FUNCTION F_CAMERA_Evaluation : BOOL
VAR_INPUT
	nExpectedResp		: INT;
	nCodesRead			: INT;
	bResetEval		  	: BOOL;
END_VAR
VAR_IN_OUT
	aCodeData			: ARRAY[1..cMAX_CAMERA_PROG_NUMBER] OF ST_CAMERA_CodeData;
	stCameraEvaluation	: ST_CAMERA_Evaluation;
END_VAR
VAR
	nImageIndex			: INT;
END_VAR

IF bResetEval THEN
	MEMSET(ADR(stCameraEvaluation), 16#00, SIZEOF(stCameraEvaluation));
	F_CAMERA_Evaluation	:= TRUE;
END_IF

(* Camera Evaluation- update total codes scanned and no-reads *)
stCameraEvaluation.nTotalReads := stCameraEvaluation.nTotalReads + F_SafeTo_UDINT(nExpectedResp);

stCameraEvaluation.nNOKCodes:= stCameraEvaluation.nNOKCodes  + F_SafeTo_UDINT(nExpectedResp - nCodesRead);
stCameraEvaluation.nReadCodes := stCameraEvaluation.nTotalReads - stCameraEvaluation.nNOKCodes;
(* scan number and determine if data will be written to primary or secondary camera data *)

(* for each pack code read *)
FOR nImageIndex := 1 TO LIMIT(1, nCodesRead, cMAX_CAMERA_PROG_NUMBER)  DO

	CASE aCodeData[nImageIndex].nEvaluation OF
		1:	stCameraEvaluation.nPoorCodes :=  stCameraEvaluation.nPoorCodes + 1;
		2:	stCameraEvaluation.nFairCodes :=  stCameraEvaluation.nFairCodes + 1;
		3:	stCameraEvaluation.nGoodCodes :=  stCameraEvaluation.nGoodCodes + 1;
	END_CASE
END_FOR

(*Pack Confirmation Camera Evaluation statistics*)
stCameraEvaluation.fReadEfficiency			:= F_SafeDIV(stCameraEvaluation.nReadCodes*100, stCameraEvaluation.nTotalReads);
stCameraEvaluation.fNOKEfficiency			:= F_SafeDIV(stCameraEvaluation.nNOKCodes*100, stCameraEvaluation.nTotalReads);

stCameraEvaluation.fGoodEfficiency		:= F_SafeDIV(stCameraEvaluation.nGoodCodes*100, ( stCameraEvaluation.nTotalReads - stCameraEvaluation.nNOKCodes));
stCameraEvaluation.fFairEfficiency		:= F_SafeDIV(stCameraEvaluation.nFairCodes*100, ( stCameraEvaluation.nTotalReads - stCameraEvaluation.nNOKCodes));
stCameraEvaluation.fPoorEfficiency		:= F_SafeDIV(stCameraEvaluation.nPoorCodes*100, ( stCameraEvaluation.nTotalReads - stCameraEvaluation.nNOKCodes));

END_FUNCTION

(* stored: Version 1.1.0.1
   POU F_CAMERA_Evaluation: Id {b763fefc-63b2-4d99-943e-1d10ad6f1ce6}, SpecialFunc None *)
